FUNCTION_BLOCK MQTTSUBSCRIBE_73D9883955B65591 (* Generic Interface Function Block Type *)
  (* Standard: 61499-2 *)
  (* Version 0.0, 05/11/2020, SESA489471, nxtControl GmBH, Template *)
  PACKAGE UAO.Hackathon;
  (* Compiler Cpp nxtControl builtin 1.0 *)
  {SET_ATTRIBUTE(Runtime.FBType.ImplementingType, nxtControl.CommProtocols#DYNGEN_MQTTSUBSCRIBE)}
  {SET_ATTRIBUTE(Configuration.GenericFBType.InterfaceParams, nxtControl.CommProtocols#CNTX:=1)}
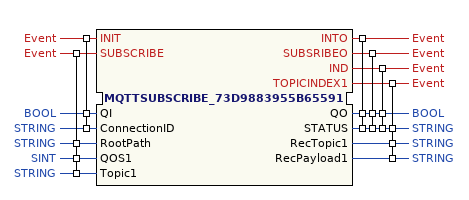
  EVENT_INPUT
    INIT WITH QI, ConnectionID; (* Request events for dedicated input data sets *)
    SUBSCRIBE WITH Topic1, QOS1, RootPath;
  END_EVENT
  EVENT_OUTPUT
    INTO WITH QO, STATUS; (* Confirmation from Resource for a dedicated request *)
    SUBSRIBEO WITH STATUS, QO; (* Indication from Resource *)
    IND WITH STATUS, QO;
    TOPICINDEX1 WITH RecPayload1, RecTopic1, STATUS;
  END_EVENT
  VAR_INPUT
    QI : BOOL;
    ConnectionID : STRING; (* MQTT Client ID *)
    RootPath : STRING;
    QOS1 : SINT; (* Quality of Service *)
    Topic1 : STRING; (* Topic to subscribe *)
  END_VAR
  VAR_OUTPUT
    QO : BOOL;
    STATUS : STRING;
    RecTopic1 : STRING;
    RecPayload1 : STRING;
  END_VAR
  EC_STATES
    START;
  END_STATES
END_FUNCTION_BLOCK
